TYPE ST_MC_Status :
STRUCT
	
	Status		: BOOL;
	Done	 	: BOOL;
	Busy	 	: BOOL;
	Error	 	: BOOL;
	Active	 	: BOOL;
	CmdAborted 	: BOOL;
	InVelocity	: BOOL;
	errorID	 	: UDINT;
	
END_STRUCT
END_TYPE

(* stored: Version 1.1.0.1, ProductVersion 3.1.4024.9
   DUT ST_MC_Status: Id {8e99dd6f-924e-4f6a-ab3a-6b49ac231634} *)
